// TwinCAT 3 PLC project Drehzahl
// ProgramVersion: 3.1.4023.0
// libraries:
//   Tc2_Standard, * (Beckhoff Automation GmbH)
//   Tc2_System, * (Beckhoff Automation GmbH)
//   Tc3_Module, * (Beckhoff Automation GmbH)
// project tree:
//   DUTs/ E_Controller_Mode.TcDUT, E_System_Mode.TcDUT, S_PID_Param.TcDUT (not stored)
//   GVLs/ GVL_Motor.TcGVL
//   / PlcTask.TcTTO
//   POUs/ FB_PID_Controller.TcPOU, MAIN.TcPOU
// real-time tasks:
//   TASK PlcTask: cycle T#10ms, priority 20, ADS port 350
// motion (NC):
//   TASK NC-Task 1 SAF: cycle T#2ms, priority 4, ADS port 501
//   TASK NC-Task 1 SVB: cycle T#10ms, priority 8, ADS port 511
//   AXIS Axis 1 (id 1)
//     OtherSettings: AllowMotionCmdToSlave=true
//     encoder EncType=4
//       EncPara: MaxCount=#x0000ffff
//         Inc: RefSoftSyncMask=#x0000ffff
//     drive DrvType=23
//       Analog: TorqueSetpointScale=10, ScaleFactorActTorque=0.1
//       TimeComp: TaskDelayCycles=1
//     controller CtrType=1
//       CtrPara: PriorControlFactor=1
//         Observer: BandWidth=20
//   AXIS Axis 2 (id 2)
//     OtherSettings: AllowMotionCmdToSlave=true
//     encoder EncType=4
//       EncPara: MaxCount=#x0000ffff
//         Inc: RefSoftSyncMask=#x0000ffff
//     drive DrvType=23
//       Analog: TorqueSetpointScale=10, ScaleFactorActTorque=0.1
//       TimeComp: TaskDelayCycles=1
//     controller CtrType=1
//       CtrPara: PriorControlFactor=1
//         Observer: BandWidth=20
// I/O:
//   DEVICE Device 1 (EtherCAT), AmsNetId 10.180.42.23.2.1
//     Term 1 (EK1200) [EK1200-5000 EtherCAT Power supply (2A E-Bus)]
//       Term 2 (EL1004) [EL1004 4Ch. Dig. Input 24V, 3ms]
//       Term 3 (EL2004) [EL2004 4Ch. Dig. Output 24V, 0.5A]
//       Term 4 (EL3004) [EL3004 4Ch. Ana. Input +/-10V]
//       Term 5 (EL4034) [EL4034 4Ch. Ana. Output +/-10V, 12bit]
//       Term 6 (EK1110) [EK1110 EtherCAT extension]
//     Term 7 (EK1100) [EK1100 EtherCAT Coupler (2A E-Bus)]
//       Term 8 (EL3004) [EL3004 4Ch. Ana. Input +/-10V]
//       Term 9 (EL5101) [EL5101 1Ch. Inc. Encoder 5V]
//       Term 10 (EL7342) [EL7342 2Ch. DC motor output stage (50V, 3.5A)]
//       Term 11 (EL9011) [EL9011 End Terminal]
// variable links:
//   NC-Task 1 SAF/Axes/Axis 1 <-> Device 1 (EtherCAT)/Term 7 (EK1100)/Term 10 (EL7342)
//     Drive/Inputs/In/nState1 @bit 3 <-> DCM Status Channel 1/Status/Error
//     Drive/Inputs/In/nState1 @bit 5 <-> DCM Status Channel 1/Status/Moving negative
//     Drive/Inputs/In/nState1 @bit 4 <-> DCM Status Channel 1/Status/Moving positive
//     Drive/Inputs/In/nState1 @bit 1 <-> DCM Status Channel 1/Status/Ready
//     Drive/Inputs/In/nState1 <-> DCM Status Channel 1/Status/Ready to enable
//     Drive/Inputs/In/nState1 @bit 6 <-> DCM Status Channel 1/Status/Torque reduced
//     Drive/Inputs/In/nState1 @bit 2 <-> DCM Status Channel 1/Status/Warning
//     Drive/Inputs/In/nState2 @bit 3 <-> DCM Status Channel 1/Status/Digital input 1
//     Drive/Inputs/In/nState2 @bit 4 <-> DCM Status Channel 1/Status/Digital input 2
//     Drive/Inputs/In/nState2 @bit 5 <-> DCM Status Channel 1/Status/Sync error
//     Drive/Inputs/In/nState2 @bit 7 <-> DCM Status Channel 1/Status/TxPDO Toggle
//     Drive/Inputs/In/nState4 @bit 1 <-> WcState/InputToggle
//     Drive/Inputs/In/nState4 <-> WcState/WcState
//     Drive/Outputs/Out/nCtrl1 @bit 2 <-> DCM Control Channel 1/Control/Reduce torque
//     Drive/Outputs/Out/nCtrl1 @bit 1 <-> DCM Control Channel 1/Control/Reset
//     Enc/Inputs/In/nDataIn1[0] <-> ENC Status compact Channel 1/Counter value
//     Enc/Inputs/In/nDataIn2[0] <-> ENC Status compact Channel 1/Latch value
//     Enc/Inputs/In/nState1 @bit 4 <-> ENC Status compact Channel 1/Status/Counter overflow
//     Enc/Inputs/In/nState1 @bit 3 <-> ENC Status compact Channel 1/Status/Counter underflow
//     Enc/Inputs/In/nState1 @bit 7 <-> ENC Status compact Channel 1/Status/Extrapolation stall
//     Enc/Inputs/In/nState1 @bit 1 <-> ENC Status compact Channel 1/Status/Latch extern valid
//     Enc/Inputs/In/nState1 @bit 2 <-> ENC Status compact Channel 1/Status/Set counter done
//     Enc/Inputs/In/nState2 @bit 4 <-> ENC Status compact Channel 1/Status/Status of extern latch
//     Enc/Inputs/In/nState2 <-> ENC Status compact Channel 1/Status/Status of input A
//     Enc/Inputs/In/nState2 @bit 1 <-> ENC Status compact Channel 1/Status/Status of input B
//     Enc/Inputs/In/nState2 @bit 5 <-> ENC Status compact Channel 1/Status/Sync error
//     Enc/Inputs/In/nState2 @bit 7 <-> ENC Status compact Channel 1/Status/TxPDO Toggle
//     Enc/Inputs/In/nState4 @bit 1 <-> WcState/InputToggle
//     Enc/Inputs/In/nState4 <-> WcState/WcState
//     Enc/Outputs/Out/nCtrl1 @bit 3 <-> ENC Control compact Channel 1/Control/Enable latch extern on negative edge
//     Enc/Outputs/Out/nCtrl1 @bit 1 <-> ENC Control compact Channel 1/Control/Enable latch extern on positive edge
//     Enc/Outputs/Out/nCtrl1 @bit 2 <-> ENC Control compact Channel 1/Control/Set counter
//     Enc/Outputs/Out/nDataOut1[0] <-> ENC Control compact Channel 1/Set counter value
//   NC-Task 1 SAF/Axes/Axis 2 <-> Device 1 (EtherCAT)/Term 7 (EK1100)/Term 10 (EL7342)
//     Drive/Inputs/In/nState1 @bit 3 <-> DCM Status Channel 2/Status/Error
//     Drive/Inputs/In/nState1 @bit 5 <-> DCM Status Channel 2/Status/Moving negative
//     Drive/Inputs/In/nState1 @bit 4 <-> DCM Status Channel 2/Status/Moving positive
//     Drive/Inputs/In/nState1 @bit 1 <-> DCM Status Channel 2/Status/Ready
//     Drive/Inputs/In/nState1 <-> DCM Status Channel 2/Status/Ready to enable
//     Drive/Inputs/In/nState1 @bit 6 <-> DCM Status Channel 2/Status/Torque reduced
//     Drive/Inputs/In/nState1 @bit 2 <-> DCM Status Channel 2/Status/Warning
//     Drive/Inputs/In/nState2 @bit 3 <-> DCM Status Channel 2/Status/Digital input 1
//     Drive/Inputs/In/nState2 @bit 4 <-> DCM Status Channel 2/Status/Digital input 2
//     Drive/Inputs/In/nState2 @bit 5 <-> DCM Status Channel 2/Status/Sync error
//     Drive/Inputs/In/nState2 @bit 7 <-> DCM Status Channel 2/Status/TxPDO Toggle
//     Drive/Inputs/In/nState4 @bit 1 <-> WcState/InputToggle
//     Drive/Inputs/In/nState4 <-> WcState/WcState
//     Drive/Outputs/Out/nCtrl1 <-> DCM Control Channel 2/Control/Enable
//     Drive/Outputs/Out/nCtrl1 @bit 2 <-> DCM Control Channel 2/Control/Reduce torque
//     Drive/Outputs/Out/nCtrl1 @bit 1 <-> DCM Control Channel 2/Control/Reset
//     Drive/Outputs/Out/nDataOut2[0] <-> DCM Velocity Channel 2/Velocity
//     Enc/Inputs/In/nDataIn1[0] <-> ENC Status compact Channel 2/Counter value
//     Enc/Inputs/In/nDataIn2[0] <-> ENC Status compact Channel 2/Latch value
//     Enc/Inputs/In/nState1 @bit 4 <-> ENC Status compact Channel 2/Status/Counter overflow
//     Enc/Inputs/In/nState1 @bit 3 <-> ENC Status compact Channel 2/Status/Counter underflow
//     Enc/Inputs/In/nState1 @bit 7 <-> ENC Status compact Channel 2/Status/Extrapolation stall
//     Enc/Inputs/In/nState1 @bit 1 <-> ENC Status compact Channel 2/Status/Latch extern valid
//     Enc/Inputs/In/nState1 @bit 2 <-> ENC Status compact Channel 2/Status/Set counter done
//     Enc/Inputs/In/nState2 @bit 4 <-> ENC Status compact Channel 2/Status/Status of extern latch
//     Enc/Inputs/In/nState2 <-> ENC Status compact Channel 2/Status/Status of input A
//     Enc/Inputs/In/nState2 @bit 1 <-> ENC Status compact Channel 2/Status/Status of input B
//     Enc/Inputs/In/nState2 @bit 5 <-> ENC Status compact Channel 2/Status/Sync error
//     Enc/Inputs/In/nState2 @bit 7 <-> ENC Status compact Channel 2/Status/TxPDO Toggle
//     Enc/Inputs/In/nState4 @bit 1 <-> WcState/InputToggle
//     Enc/Inputs/In/nState4 <-> WcState/WcState
//     Enc/Outputs/Out/nCtrl1 @bit 3 <-> ENC Control compact Channel 2/Control/Enable latch extern on negative edge
//     Enc/Outputs/Out/nCtrl1 @bit 1 <-> ENC Control compact Channel 2/Control/Enable latch extern on positive edge
//     Enc/Outputs/Out/nCtrl1 @bit 2 <-> ENC Control compact Channel 2/Control/Set counter
//     Enc/Outputs/Out/nDataOut1[0] <-> ENC Control compact Channel 2/Set counter value
//   Drehzahl/Drehzahl Instance <-> Device 1 (EtherCAT)/Term 7 (EK1100)/Term 10 (EL7342)
//     PlcTask Outputs/GVL_Motor.MotorEnable <-> DCM Control Channel 1/Control/Enable
//     PlcTask Outputs/GVL_Motor.MotorVelocity <-> DCM Velocity Channel 1/Velocity
//   Drehzahl/Drehzahl Instance <-> Device 1 (EtherCAT)/Term 7 (EK1100)/Term 9 (EL5101)
//     PlcTask Inputs/GVL_Motor.CounterOverflow <-> ENC Status compact/Status/Counter overflow
//     PlcTask Inputs/GVL_Motor.CounterUnderflow <-> ENC Status compact/Status/Counter underflow
//     PlcTask Inputs/GVL_Motor.MotorPosition <-> ENC Status compact/Counter value

CONFIGURATION Drehzahl
    RESOURCE PLC ON TwinCAT3
        TASK PlcTask(INTERVAL := T#10ms, PRIORITY := 20);
        PROGRAM MAIN WITH PlcTask : MAIN;
    END_RESOURCE
END_CONFIGURATION

// ---- DUTs/E_Controller_Mode.TcDUT
{attribute 'qualified_only'}
{attribute 'strict'}
TYPE E_Controller_Mode :
(
	Controller_Init:= 0,
	Controller_OpenLoop, 
	Controller_ClosedLoop
	
);
END_TYPE

// ---- DUTs/E_System_Mode.TcDUT
{attribute 'qualified_only'}
{attribute 'strict'}
TYPE E_System_Mode :
(
	System_Init := 0,
	System_Run

);
END_TYPE

// ---- GVLs/GVL_Motor.TcGVL
{attribute 'qualified_only'}
VAR_GLOBAL
    
	MotorPosition  		AT %I* : UINT;
	CounterOverflow 	AT %I* : BOOL;
	CounterUnderflow 	AT %I* : BOOL;
	MotorEnable			AT %Q* : BOOL;
	MotorVelocity 		AT %Q* : INT;
	
END_VAR

// ---- POUs/MAIN.TcPOU
PROGRAM MAIN
VAR
	LastMotorPosition	: 	UINT;
	Difference			:	INT;
	DrehzahlRpm			: 	REAL;
	DrehzahlRps			: 	REAL;
	DrehzahlRef			:   REAL;
	OverflowCalculated	: 	BOOL := FALSE;
	UnderflowCalculated	: 	BOOL := FALSE;
	VoltageMotor		:   REAL;
	ModeController		:   E_Controller_Mode := 0;
	Mode				:	E_System_Mode;
	PID					: 	FB_PID_Controller;
	PID_Param			:   S_PID_Param;
END_VAR
VAR CONSTANT
	cycleTimeS			:	REAL := 0.01;
	ImpulsePerRevolution: 	UINT := 2048; 
	uintUpperBound		: 	UINT := 65535;
	MaxVelocity			: 	INT := 32767;
	MaxVoltage			:   REAL := 24;
END_VAR

// calculate drehzahl
Difference := UINT_TO_INT(GVL_MOTOR.MotorPosition-LastMotorPosition);
// handle overflow / underflow
IF GVL_MOTOR.CounterOverflow AND OverflowCalculated = FALSE THEN
	OverflowCalculated := TRUE;
	Difference := UINT_TO_INT((uintUpperBound - LastMotorPosition) + GVL_MOTOR.MotorPosition);
ELSIF GVL_MOTOR.CounterOverflow = FALSE THEN   // reset flag
	OverflowCalculated := FALSE;
END_IF
IF GVL_MOTOR.CounterUnderflow AND UnderflowCalculated = FALSE THEN
	UnderflowCalculated := TRUE;
	Difference := UINT_TO_INT((GVL_MOTOR.MotorPosition - uintUpperBound) - LastMotorPosition);
ELSIF GVL_MOTOR.CounterUnderflow = FALSE THEN   // reset flag
	UnderflowCalculated := FALSE;
END_IF
DrehzahlRps := Difference / (cycleTimeS * ImpulsePerRevolution);
DrehzahlRpm := DrehzahlRps * 60;
// store values
LastMotorPosition := GVL_MOTOR.MotorPosition;

IF VoltageMotor = 0 THEN
	GVL_Motor.MotorVelocity := 0;
ELSE		
	GVL_Motor.MotorVelocity := REAL_TO_INT(VoltageMotor / MaxVoltage * MaxVelocity);	
END_IF
CASE ModeController OF
	E_Controller_Mode.Controller_Init:
		PID_Param.Kp 	:= 0.0096;
		PID_Param.Ti 	:= 0.11;
		PID_Param.Td 	:= 0.0275;
		PID_Param.Tr 	:= SQRT(PID_Param.Ti*PID_Param.Td);
		PID_Param.N  	:= 20;
		PID_Param.ARW	:= TRUE;
		PID_Param.umax:= 20;
		PID_Param.umin:= -20;
		Mode := E_System_Mode.System_Init;
		PID(ref:=0, y:=0, Mode := Mode, Param:=PID_Param, T:=cycleTimeS);
		GVL_MOTOR.MotorEnable := TRUE;
	;
	
	E_Controller_Mode.Controller_OpenLoop:

	;
	
	E_Controller_Mode.Controller_ClosedLoop:
		Mode := E_System_Mode.System_Run;
		PID(ref:=DrehzahlRef, y:=DrehzahlRpm, Mode := Mode, Param:=PID_Param, T:=cycleTimeS);
		VoltageMotor := PID.u_sat;
	;
	
END_CASE

END_PROGRAM

// ---- POUs/FB_PID_Controller.TcPOU
FUNCTION_BLOCK FB_PID_Controller
VAR_INPUT
	ref		: REAL;		// Aktuelle Referenzgroesse (Soll-Groesse)
	y		: REAL;		// Aktuelle Regelgroesse (Ist-Groesse)
	Mode	: E_System_Mode; 	// Aktueller Modus
	Param	: S_PID_Param;		// PID Regler Parameter
	T		: REAL;				// Abtastzeit
END_VAR
VAR_OUTPUT
	u_k		: REAL; 			// Ausgangsgroesse
	u_sat	: REAL; 			// Ausgangsgroesse gesaettigt
END_VAR
VAR
	e_k 	: REAL;
	e_k_1	: REAL;
	u_p		: REAL;
	u_d		: REAL;
	u_d_k_1	: REAL;
	u_i_k_1	: REAL;
	u_aw	: REAL;				// anti reset windup back calculation result
	bi		: REAL;				// calculation parameter for I term
	bd		: REAL;				// calculation parameter for D term
	ad		: REAL;				// calculation parameter for D term
	
END_VAR

CASE Mode OF
	E_System_Mode.System_Init:
		// calculate coefficients
		bi := Param.Kp * T / (2*Param.Ti);
		ad := Param.Td / (Param.Td + Param.N * T);
		bd := (Param.Kp * Param.N * Param.Td) / (Param.Td + Param.N * T);
		
		// reset values
		u_i_k_1	:= 0;
		u_d_k_1	:= 0;
		e_k_1	:= 0;
		u_aw	:= 0;
		
	E_System_Mode.System_Run:
		// implements differencial equation
		
		// compute the error
		e_k := ref - y;
		
		// proportinal term
		u_p := Param.Kp * e_k;
		
		// derivative term with filter
		u_d	:= ad * u_d_k_1 + bd * (e_k - e_k_1);
	
		// total command (u_i from last cycle since it gets calculated later)
		u_k := u_p + u_i_k_1 + u_d;
		
		// saturation
		u_sat := u_k;
		IF u_k > Param.umax THEN
			u_sat := Param.umax;
		ELSIF u_k < Param.umin THEN
			u_sat := Param.umin;
		END_IF
		
		// anti reset windup for next loop
		IF Param.ARW THEN
			u_aw := (T/Param.Tr) * (u_sat - u_k);
		ELSE
			u_aw := 0;
		END_IF
		
		// integral term (Trapezregel)
		u_i_k_1 := u_i_k_1 + bi * (e_k + e_k_1) + u_aw;
		
		// store vars for next step
		u_d_k_1 := u_d;
		e_k_1 := e_k;
		
	ELSE  // default assignment
	;
		
END_CASE

END_FUNCTION_BLOCK
